Staubli VAL3: cartesianSpace.dtx

public pointRx cCartesianPos = {fatherId=world[0]}
public CartesianVel cCartesianVel
  [0]
    num vx
    num vy
    num vz
    num vrx
    num vry
    num vrz
public CartesianAccel cCartesianAccel
  [0]
    num ax
    num ay
    num az
    num arx
    num ary
    num arz
public CartesianForce cCartesianForce
  [0]
    num fx
    num fy
    num fz
    num frx
    num fry
    num frz
